Universal Robots PolyScope program: b_mbase2.urp

Program b_mbase2 (installation=default directory=/programs/Burkat_U_Plant createdIn=5.12.6.1102099 lastSavedIn=5.12.6.1102099 robotSerialNumber=20215500597)
Calibrated DH parameters: a=[0.000193, -0.066673, -0.391568, -0.000012, 0.00005, 0]; d=[0.162643, -472.05677, 465.132521, 7.058239, 0.099746, 0.099582]; alpha=[1.571116, 0.00089, 0.003862, 1.569269, -1.569248, 0]; deltaTheta=[0, -1.413394, 7.628392, 0.068187, 0, -0.000001]
Robot Program (runOnlyOnce=true)
  MoveJ speed 60 deg/s, acceleration 80 deg/s^2 (useActiveTCP=true) feature=Base
    Waypoint Waypoint_19: TCP in base x=-66.326 y=-841.615 z=276.687 mm, rx=1.6517 ry=-0.0259 rz=-0.093 rad; joints [71.48, -64.638, 86.648, -17.383, 75.945, -3.629] deg; TCP offset x=0 y=0 z=191.5 mm, rx=0 ry=0 rz=0 rad
